(* IEC 61131-3 sources: website/app/projektit/rau-tyokalut/modbusrajapinta/examples/Common_functions, 30 files *)

(* ---- bitClearF.ST ---- *)
FUNCTION bitClearF : BOOL
VAR_INPUT
bitString : word;
bitNumber : uint;
END_VAR

VAR
bResult : bool;
wTemp : word;
END_VAR
(************************************************************)
(*	Function checks if bit is cleared in given bit string 	*)
(*															*)
(*	Inputs: bitString as 16bit word							*)
(*			bitNumber as unsigned integer from 0 to 15		*)
(*	Returns: Boolean value							  		*)
(*	Use: if bitClearF(bitString, bitNumber) then	 	  	*)
(*				do_something();						  		*)
(*		 end_if;											*)
(*													  		*)
(************************************************************)

if bitNumber > 15 then
	bResult := false;
else
	wTemp := 1;
	wTemp := SHL(wTemp, bitNumber);
	bResult := (bitString AND wTemp) = 0;
end_if;
bitClearF := bResult;

END_FUNCTION

(* ---- bitSetF.ST ---- *)
FUNCTION bitSetF : BOOL
VAR_INPUT
bitString : word;
bitNumber : uint;
END_VAR

VAR
bResult : bool;
wTemp : word;
END_VAR
(************************************************************)
(*	Function checks if bit is set in given bit string 		*)
(*															*)
(*	Inputs: bitString as 16bit word							*)
(*			bitNumber as unsigned integer from 0 to 15		*)
(*	Returns: Boolean value							  		*)
(*	Use: if bitSetF(bitString, bitNumber) then	 	  		*)
(*				do_something();						  		*)
(*		 end_if;											*)
(*													  		*)
(************************************************************)

if bitNumber > 15 then
	bResult := false;
else
	wTemp := 1;
	wTemp := SHL(wTemp, bitNumber);
	bResult := (bitString AND wTemp) > 0;
end_if;
bitSetF := bResult;

END_FUNCTION

(* ---- clearBitF.ST ---- *)
FUNCTION clearBitF : WORD
VAR_INPUT
bitString : word;
bitNumber : uint;
END_VAR

VAR
wResult : word;
wTemp : word;
END_VAR
(************************************************************)
(*	Function clears bit in given bit string 				*)
(*															*)
(*	Inputs: bitString as 16bit word							*)
(*			bitNumber as unsigned integer from 0 to 15		*)
(*	Returns: bitString with the bit cleared as 16bit word  	*)
(*	Use: bitString:=clearBitF(bitString, bitNumber);	 	*)
(*													  		*)
(************************************************************)

if bitNumber > 15 then
	wResult := bitString;
else
	wTemp := 1;
	wTemp := SHL(wTemp, bitNumber);
	wResult := bitString AND (16#FFFF XOR wTemp);
end_if;
clearBitF := wResult;

END_FUNCTION

(* ---- CoilF.ST ---- *)
FUNCTION CoilF : WORD
VAR_INPUT
	id_String : string(30);
	RegValue : word;
	BitMask : word;
END_VAR

VAR
	iTemp : int;
	iLockState : int;
	bFX2020 : bool;
	bReg : bool;
	ReturnValue : word;
END_VAR

bFX2020 := INT_TO_BOOL(GetDigitalPointF(Name:=id_String));
bReg:=WORD_TO_BOOL(RegValue AND BitMask);
iLockState:=GetLockStateF(Name:=id_String);

ReturnValue := RegValue;
IF id_String <> '' THEN
	if bFX2020 = bReg then
		(* Same value -> release manual override *)
		iTemp:=SetDigitalPointF(Value:=BOOL_TO_INT(bReg), LockState := 3, Name := id_String);
	elsif (iLockState = 2 or iLockState = 12) then
		(* The value have been changed in FX *)
		if (bFX2020 = true) then
			ReturnValue := (RegValue OR BitMask);
		else
			ReturnValue := (RegValue AND NOT(BitMask));
		end_if;
	else
		(* The value may have been changed in handterminal *)
	 	iTemp:=SetDigitalPointF(Value:=BOOL_TO_INT(bReg), LockState := 1, Name := id_String);
	end_if;
END_IF;

CoilF := ReturnValue;

END_FUNCTION

(* ---- CoilF_2.ST ---- *)
FUNCTION CoilF_2 : WORD
VAR_INPUT
	id_String : string(30);
	RegValue : word;
	BitMask : word;
	force : int;
END_VAR

VAR
	iTemp : int;
	iLockState : int;
	bFX2020 : bool;
	bReg : bool;
	ReturnValue : word;
END_VAR
(*Different version of the CoilF-function, added a new input parameter 'force' that indicates if the value is wanted to be
 forced from FX to the modbus device 0 = no forcing, 1 = value is forced *)

bFX2020 := INT_TO_BOOL(GetDigitalPointF(Name:=id_String));
bReg:=WORD_TO_BOOL(RegValue AND BitMask);
iLockState:=GetLockStateF(Name:=id_String);

ReturnValue := RegValue;
IF id_String <> '' THEN
	if bFX2020 = bReg then
		(* Same value -> release manual override *)
		iTemp:=SetDigitalPointF(Value:=BOOL_TO_INT(bReg), LockState := 3, Name := id_String);
	elsif (iLockState = 2 or iLockState = 12 or force = 1) then
		(* The value have been changed in FX, or user wants to force the point from FX *)
		if (bFX2020 = true) then
			ReturnValue := (RegValue OR BitMask);
		else
			ReturnValue := (RegValue AND NOT(BitMask));
		end_if;
	else
		(* The value may have been change in handterminal *)
	 	iTemp:=SetDigitalPointF(Value:=BOOL_TO_INT(bReg), LockState := 1, Name := id_String);
	end_if;
END_IF;

CoilF_2 := ReturnValue;

END_FUNCTION

(* ---- CoilF_3.ST ---- *)
FUNCTION CoilF_3 : WORD
VAR_INPUT
	id_String : string(30);
	RegValue : word;
	BitMask : word;
	Force : bool;
	ReleaseOverride : bool;
END_VAR

VAR
	iTemp : int;
	iLockState : int;
	bFX2020 : bool;
	bReg : bool;
	ReturnValue : word;
END_VAR

bFX2020 := INT_TO_BOOL(GetDigitalPointF(Name:=id_String));
bReg:=WORD_TO_BOOL(RegValue AND BitMask);
iLockState:=GetLockStateF(Name:=id_String);

ReturnValue := RegValue;
IF id_String <> '' THEN
	if bFX2020 = bReg and releaseOverride = true then
		(* Same value -> release manual override *)
		iTemp:=SetDigitalPointF(Value:=BOOL_TO_INT(bReg), LockState := 3, Name := id_String);
	elsif (iLockState = 2 or iLockState = 12 or force = true) then
		(* The value have been changed in FX *)
		if (bFX2020 = true) then
			ReturnValue := (RegValue OR BitMask);
		else
			ReturnValue := (RegValue AND NOT(BitMask));
		end_if;
	else
		(* The value may have been changed in handterminal *)
	 	iTemp:=SetDigitalPointF(Value:=BOOL_TO_INT(bReg), LockState := 1, Name := id_String);
	end_if;
END_IF;

CoilF_3 := ReturnValue;

END_FUNCTION

(* ---- DiscreteInputF.ST ---- *)
FUNCTION DiscreteInputF : INT
VAR_INPUT
	id_String : string(30);
	RegValue : word;
	BitMask : word;
END_VAR

VAR
	tulos : int;
END_VAR

IF id_String <> '' THEN
	(* Check BitMask defined bit status *)
	tulos := SetDigitalPointF(Value:=BOOL_TO_INT(WORD_TO_BOOL(RegValue AND BitMask)), LockState:=1, Name:=id_String);
	DiscreteInputF := 0;
ELSE
	DiscreteInputF := 9999;
END_IF;

END_FUNCTION

(* ---- DOUBLEHOLDINGREGF.ST ---- *)
FUNCTION DOUBLEHOLDINGREGF : UDINT
VAR_INPUT
	id_String : string(30);
	HighRegValue : word;
	LowRegValue : word;
	rMultiplier : real;
END_VAR

VAR
	rMultiply : real;
	rFX2025 : real;
	rReg : real;
	iLockState : int;
	iTemp : int;
	iReg : int;
	udiConversion : udint;
	diConversion : dint;
	rconversion : real;
	Result : int;
END_VAR
(* Zero division not allowed *)
rMultiply := rMultiplier;
if (rMultiply = 0.0) then
	rMultiply := 1.0;
end_if;

(* Read current FX2025 value *)
rFX2025 := GetAnalogPointF(Name:=id_String);

(* Convert double register value to real value *)
udiConversion := 65536*WORD_TO_UDINT(HighRegValue) + WORD_TO_UDINT(LowRegValue);
diConversion := UDINT_TO_DINT(udiConversion);
rConversion := DINT_TO_REAL(diConversion)/rMultiply;

(* Check LockState *)
iLockState:=GetLockStateF(Name:=id_String);

if id_String <> '' then
	if (rFX2025 = rConversion) then
		(* Same value -> release manual override *)
		Result := SetAnalogPointF(Value:=rConversion, LockState:=3, Name:=id_String);
	elsif (iLockState = 2 or iLockState = 12) then
		(* The value have been changed in FX *)
		diConversion := REAL_TO_DINT(rFX2025 * rMultiply);
		udiConversion := DINT_TO_UDINT(diConversion);
	else
		(* The value may have been changed in modbus equipment *)
		Result := SetAnalogPointF(Value:=rConversion, LockState:=1, Name:=id_String);
	end_if;
end_if;

DoubleHoldingRegF := udiConversion;

END_FUNCTION

(* ---- DOUBLEHOLDINGREGF_3DINT.ST ---- *)
FUNCTION DOUBLEHOLDINGREGF_3DINT : UDINT
VAR_INPUT
	id_String : string(30);
	HighRegValue : word;
	LowRegValue : word;
	rMultiplier : real;
	Force : bool;
	ReleaseOverride : bool;
END_VAR

VAR
	rMultiply : real;
	rFX2025 : real;
	rReg : real;
	iLockState : int;
	iTemp : int;
	iReg : int;
	udiConversion : udint;
	diConversion : dint;
	rconversion : real;
	Result : int;
END_VAR
(* Zero division not allowed *)
rMultiply := rMultiplier;
if (rMultiply = 0.0) then
	rMultiply := 1.0;
end_if;

(* Read current FX2025 value *)
rFX2025 := GetAnalogPointF(Name:=id_String);

(* Convert double register value to real value *)
udiConversion := 65536*WORD_TO_UDINT(HighRegValue) + WORD_TO_UDINT(LowRegValue);
diConversion := UDINT_TO_DINT(udiConversion);
rConversion := DINT_TO_REAL(diConversion)/rMultiply;

(* Check LockState *)
iLockState:=GetLockStateF(Name:=id_String);

if id_String <> '' then
	if (rFX2025 = rConversion and ReleaseOverride = true) then
		(* Same value -> release manual override *)
		Result := SetAnalogPointF(Value:=rConversion, LockState:=3, Name:=id_String);
	elsif (iLockState = 2 or iLockState = 12 or Force = true) then
		(* The value have been changed in FX *)
		diConversion := REAL_TO_DINT(rFX2025 * rMultiply);
		udiConversion := DINT_TO_UDINT(diConversion);
	else
		(* The value may have been changed in modbus equipment *)
		Result := SetAnalogPointF(Value:=rConversion, LockState:=1, Name:=id_String);
	end_if;
end_if;

DoubleHoldingRegF_3DINT := udiConversion;

END_FUNCTION

(* ---- DOUBLEHOLDINGREGF_3UDINT.ST ---- *)
FUNCTION DOUBLEHOLDINGREGF_3UDINT : UDINT
VAR_INPUT
	id_String : string(30);
	HighRegValue : word;
	LowRegValue : word;
	rMultiplier : real;
	Force : bool;
	ReleaseOverride : bool;
END_VAR

VAR
	rMultiply : real;
	rFX2025 : real;
	rReg : real;
	iLockState : int;
	iTemp : int;
	iReg : int;
	udiConversion : udint;
	rconversion : real;
	Result : int;
END_VAR
(* Zero division not allowed *)
rMultiply := rMultiplier;
if (rMultiply = 0.0) then
	rMultiply := 1.0;
end_if;

(* Read current FX2025 value *)
rFX2025 := GetAnalogPointF(Name:=id_String);

(* Convert double register value to real value *)
udiConversion := 65536*WORD_TO_UDINT(HighRegValue) + WORD_TO_UDINT(LowRegValue);
rConversion := UDINT_TO_REAL(udiConversion)/rMultiply;

(* Check LockState *)
iLockState:=GetLockStateF(Name:=id_String);

if id_String <> '' then
	if (rFX2025 = rConversion and ReleaseOverride = true) then
		(* Same value -> release manual override *)
		Result := SetAnalogPointF(Value:=rConversion, LockState:=3, Name:=id_String);
	elsif (iLockState = 2 or iLockState = 12 or Force = true) then
		(* The value have been changed in FX *)
		udiConversion := REAL_TO_UDINT(rFX2025 * rMultiply);
	else
		(* The value may have been changed in modbus equipment *)
		Result := SetAnalogPointF(Value:=rConversion, LockState:=1, Name:=id_String);
	end_if;
end_if;

DoubleHoldingRegF_3UDINT := udiConversion;

END_FUNCTION

(* ---- DoubleHoldingRegF_EM.ST ---- *)
FUNCTION DoubleHoldingRegF_EM : UDINT
VAR_INPUT
	id_String : string(30);
	HighRegValue : word;
	LowRegValue : word;
	rMultiplier : real;
END_VAR

VAR
	rMultiply : real;
	rFX2025 : real;
	rReg : real;
	iLockState : int;
	iTemp : int;
	iReg : int;
	udiConversion : udint;
	diConversion : dint;
	rconversion : real;
	Result : int;
END_VAR
(* Zero division not allowed *)
rMultiply := rMultiplier;
if (rMultiply = 0.0) then
	rMultiply := 1.0;
end_if;

(* Read current FX2025 value *)
rFX2025 := GetAnalogPointF(Name:=id_String);

(* Convert double register value to real value *)
udiConversion := 65536*WORD_TO_UDINT(HighRegValue) + WORD_TO_UDINT(LowRegValue);
diConversion := UDINT_TO_DINT(udiConversion);
rConversion := DINT_TO_REAL(diConversion)/rMultiply;

(* Check LockState *)
iLockState:=GetLockStateF(Name:=id_String);

if id_String <> '' then
	if (rFX2025 = rConversion) then
		(* Same value -> release manual override *)
		Result := SetAnalogPointF(Value:=rConversion, LockState:=3, Name:=id_String);
	elsif (iLockState = 2 or iLockState = 12) then
		(* The value have been changed in FX *)
		(* Energiamittarin rekisterit voidaan vain nollata *)
		if (rFX2025 <> 0.0) then
			Result := SetAnalogPointF(Value:=rConversion, LockState:=3, Name:=id_String);
		else
			udiConversion := 0;
		end_if;
	else
		(* The value may have been changed in modbus equipment *)
		Result := SetAnalogPointF(Value:=rConversion, LockState:=1, Name:=id_String);
	end_if;
end_if;

DoubleHoldingRegF_EM := udiConversion;

END_FUNCTION

(* ---- DoubleHoldingRegF_FLOAT.ST ---- *)
FUNCTION DoubleHoldingRegF_FLOAT : DWORD
VAR_INPUT
	id_String : string(30);
	LowRegValue : word;
	HighRegValue : word;
END_VAR

VAR
	rFX2020 : real;
	rReg : real;
	iLockState : int;
	iTemp : int;
	iReg : int;
	dwArvo : dword;
	realArvo : real;
END_VAR
(*point value in Fx*)
rFX2020 := GetAnalogPointF(Name:=id_String);

(* Value from modbus *)
dwArvo := WORD_TO_DWORD( HighRegValue );  (* Muunnnos 32 bittiseksi *)
dwArvo := SHL( dwArvo, 16 );   (* Siirret??n 16 bitti? vasemmalle *)
dwArvo := dwArvo OR WORD_TO_DWORD( LowRegValue );   (* Lis?t??n alemmat 16 bitti? *)
realArvo := WORD2_TO_REAL( dwArvo )  ;   (* Muunnetaan REAL tyyppiseksi *)
iLockState:=GetLockStateF(Name:=id_String);

IF id_String <> '' THEN
	if rFX2020 = realArvo then
		(* Same value -> release manual override *)
		iTemp:=SetAnalogPointF(Value:=rReg, LockState := 3, Name := id_String);
	elsif (iLockState = 2 or iLockState = 12) then
		(* The value have been changed in FX *)
		realArvo := rFX2020;
		dwArvo := REAL_TO_WORD2(realArvo); (*modify the return value so that it can be written to registers*)
	else
		(* The value may have been change in handterminal *)
		iTemp:=SetAnalogPointF(Value:=realArvo, LockState := 1, Name := id_String);
	end_if;
END_IF;

(* return the register values in a DWORD*)
DoubleHoldingRegF_FLOAT := dwArvo;

END_FUNCTION

(* ---- DoubleInputReg_Float.ST ---- *)
FUNCTION DoubleInputReg_Float : REAL
VAR_INPUT
	id_String : string(30);
	HighRegValue : word;
	LowRegValue : word;
END_VAR

VAR
	dwArvo : dword;
	realArvo : real;
	result : int;
END_VAR

dwArvo := WORD_TO_DWORD( HighRegValue );  (* Muunnnos 32 bittiseksi *)
dwArvo := SHL( dwArvo, 16 );   (* Siirret??n 16 bitti? vasemmalle *)
dwArvo := dwArvo OR WORD_TO_DWORD( LowRegValue );   (* Lis?t??n alemmat 16 bitti? *)
realArvo := WORD2_TO_REAL( dwArvo )  ;   (* Muunnetaan REAL tyyppiseksi *)

(* Talletetaan arvo mittauspisteeseen *)
result := SetAnalogPointF( Value := realArvo , LockState:=1, Name:= id_String );

DoubleInputReg_Float := realArvo;

END_FUNCTION

(* ---- DoubleInputReg_Float_jakaja.ST ---- *)
FUNCTION DoubleInputReg_Float_jakaja : REAL
VAR_INPUT
	id_String : string(30);
	HighRegValue : word;
	LowRegValue : word;
	jakaja : real;
END_VAR

VAR
	dwArvo : dword;
	realArvo : real;
	result : int;
END_VAR

dwArvo := WORD_TO_DWORD( HighRegValue );  (* Muunnnos 32 bittiseksi *)
dwArvo := SHL( dwArvo, 16 );   (* Siirret??n 16 bitti? vasemmalle *)
dwArvo := dwArvo OR WORD_TO_DWORD( LowRegValue );   (* Lis?t??n alemmat 16 bitti? *)
realArvo := WORD2_TO_REAL( dwArvo )  ;   (* Muunnetaan REAL tyyppiseksi *)

if(jakaja > 0.0) then
	realArvo := realArvo / jakaja;
end_if;

(* Talletetaan arvo mittauspisteeseen *)
result := SetAnalogPointF( Value := realArvo , LockState:=1, Name:= id_String );

DoubleInputReg_Float_jakaja := realArvo;

END_FUNCTION

(* ---- DoubleInputReg_WM14.ST ---- *)
FUNCTION DoubleInputReg_WM14 : REAL
VAR_INPUT
	id_String : string(30);
	HighRegValue : word;
	LowRegValue : word;
END_VAR

VAR
	dwArvo : dword;
	realArvo : real;
	result : int;
END_VAR

dwArvo := WORD_TO_DWORD( HighRegValue );  (* Muunnnos 32 bittiseksi *)
dwArvo := SHL( dwArvo, 16 );   (* Siirret??n 16 bitti? vasemmalle *)
dwArvo := dwArvo OR WORD_TO_DWORD( LowRegValue );   (* Lis?t??n alemmat 16 bitti? *)
realArvo := WORD2_TO_REAL( dwArvo )  ;   (* Muunnetaan REAL tyyppiseksi *)

(* Talletetaan arvo mittauspisteeseen *)
result := SetAnalogPointF( Value := realArvo , LockState:=1, Name:= id_String );

DoubleInputReg_WM14 := realArvo;

END_FUNCTION

(* ---- DoubleInputRegF.ST ---- *)
FUNCTION DoubleInputRegF : UDINT
VAR_INPUT
	id_String : string(30);
	HighRegValue : word;
	LowRegValue : word;
	rMultiplier : real;
END_VAR

VAR
	rMultiply : real;
	rFX2025 : real;
	rReg : real;
	iLockState : int;
	iTemp : int;
	iReg : int;
	udiConversion : udint;
	diConversion : dint;
	rconversion : real;
	Result : int;
END_VAR
(* Zero division not allowed *)
rMultiply := rMultiplier;
if (rMultiply = 0.0) then
	rMultiply := 1.0;
end_if;

(* Convert double register value to real value *)
udiConversion := 65536*WORD_TO_UDINT(HighRegValue) + WORD_TO_UDINT(LowRegValue);
diConversion := UDINT_TO_DINT(udiConversion);
rConversion := DINT_TO_REAL(diConversion)/rMultiply;

(* Save value to point database *)
Result := SetAnalogPointF(Value:=rConversion, LockState:=1, Name:=id_String);

DoubleInputRegF := udiConversion;

END_FUNCTION

(* ---- DoubleInputRegF_DINT.ST ---- *)
FUNCTION DoubleInputRegF_DINT : UDINT
VAR_INPUT
	id_String : string(30);
	HighRegValue : word;
	LowRegValue : word;
	rMultiplier : real;
END_VAR

VAR
	rMultiply : real;
	rFX2025 : real;
	rReg : real;
	iLockState : int;
	iTemp : int;
	iReg : int;
	udiConversion : udint;
	diConversion : dint;
	rconversion : real;
	Result : int;
END_VAR
(* Zero division not allowed *)
rMultiply := rMultiplier;
if (rMultiply = 0.0) then
	rMultiply := 1.0;
end_if;

(* Convert double register value to real value *)
udiConversion := 65536*WORD_TO_UDINT(HighRegValue) + WORD_TO_UDINT(LowRegValue);
diConversion := UDINT_TO_DINT(udiConversion);
rConversion := DINT_TO_REAL(diConversion)/rMultiply;

(* Save value to point database *)
Result := SetAnalogPointF(Value:=rConversion, LockState:=1, Name:=id_String);

DoubleInputRegF_DINT := udiConversion;

END_FUNCTION

(* ---- DoubleInputRegF_UDINT.ST ---- *)
FUNCTION DoubleInputRegF_UDINT : UDINT
VAR_INPUT
	id_String : string(30);
	HighRegValue : word;
	LowRegValue : word;
	rMultiplier : real;
END_VAR

VAR
	rMultiply : real;
	rFX2025 : real;
	rReg : real;
	iLockState : int;
	iTemp : int;
	iReg : int;
	udiConversion : udint;
	rconversion : real;
	Result : int;
END_VAR
(* Zero division not allowed *)
rMultiply := rMultiplier;
if (rMultiply = 0.0) then
	rMultiply := 1.0;
end_if;

(* Convert double register value to real value *)
udiConversion := 65536*WORD_TO_UDINT(HighRegValue) + WORD_TO_UDINT(LowRegValue);
rConversion := UDINT_TO_REAL(udiConversion)/rMultiply;

(* Save value to point database *)
Result := SetAnalogPointF(Value:=rConversion, LockState:=1, Name:=id_String);

DoubleInputRegF_UDINT := udiConversion;

END_FUNCTION

(* ---- fxe_Input64F.ST ---- *)
FUNCTION fxe_Input64F :REAL
(*
PLC: Fidelix
Company: Fidelix Sverige AB
Created by: Åke Kindmark_PC2
Program: fxe_Input64F

Date		| Version	|Created under	| Changed by		| Remark
----------------------------------------------------------------------------
2021-10-07		|   		|OpenPCSv 7.1.5	| Åke Kindmark_PC2		|
*)
VAR_INPUT
	PointId						:STRING(30) := '';
	LowReg0Value				:WORD;
	LowReg1Value				:WORD;
	HighReg2Value				:WORD;
	HighReg3Value				:WORD;
	Options						:DWORD;
END_VAR

VAR
	LReg0Value					:WORD;
	LReg1Value					:WORD;
	HReg2Value					:WORD;
	HReg3Value					:WORD;
	L0_org						:WORD;
	L1_org						:WORD;
	H2_org						:WORD;
	H3_org						:WORD;
	byte1						:WORD;
	byte2						:WORD;
	byte3						:WORD;
	byte4						:WORD;
	byte5						:WORD;
	byte6						:WORD;
	byte7						:WORD;
	byte8						:WORD;
	L0_inv						:WORD;
	L1_inv						:WORD;
	H2_inv						:WORD;
	H3_inv						:WORD;
	rReg_0						:REAL;
	rReg_1						:REAL;
	rReg_2						:REAL;
	rReg_3						:REAL;
	rValue						:REAL;
	iResult						:INT;
	rMultiplier					:REAL;
	iAccess						:INT;
	iSize						:INT;
	bBitMask					:BOOL;
	bInvert						:BOOL;
	bEndian						:BOOL;
	bByte						:BOOL;
	bWord						:BOOL;
	bUnsigned					:BOOL;
END_VAR
(* Extract multiplier from options *)
CASE DWORD_TO_INT(7 AND SHR(Options, 13)) OF
	1: rMultiplier := 10.0;
	2: rMultiplier := 100.0;
	3: rMultiplier := 1000.0;
ELSE
	rMultiplier := 1.0;
END_CASE;

(* Extract access from options *)
iAccess := DWORD_TO_INT(3 AND Options);
(* Extract size from options *)
iSize := DWORD_TO_INT(SHR(Options, 11));
(* Extract bitmask flag from options *)
bBitMask := DWORD_TO_INT(16 AND Options) = 16;
(* Extract invert flag from options *)
bInvert := DWORD_TO_INT(32 AND Options) = 32;
(* Extract litle endian flag from options *)
bEndian := DWORD_TO_INT(64 AND Options) = 64;
(* Extract byte swap flag from options *)
bByte := DWORD_TO_INT(128 AND Options) = 128;
(* Extract word swap flag from options *)
bWord := DWORD_TO_INT(256 AND Options) = 256;
(* Extract unsigned flag from options *)
bUnsigned := DWORD_TO_INT(512 AND Options) = 512;

(* Read 64(4x16)-bits registervalue *)
LReg0Value := LowReg0Value;
LReg1Value := LowReg1Value;
HReg2Value := HighReg2Value;
HReg3Value := HighReg3Value;

(* Byteswap. Shift High(MSP) and Low(LSP) Bytes of each 16-bit register value? *)
IF bByte THEN
	(* Read the original value of the registers, the bytes of which are inverted *)
	L0_org := LReg0Value;
	L1_org := LReg1Value;
	H2_org := HReg2Value;
	H3_org := HReg3Value;
	(* Masking, followed by only the last 8 bits of the word *)
	byte1 := (L0_org AND 16#00FF);
	byte3 := (L1_org AND 16#00FF);
	byte5 := (H2_org AND 16#00FF);
	byte7 := (H3_org AND 16#00FF);
	(* Move the second byte to the first position, i.e. 8 bits to the left *)
	byte1 := SHL(byte1, 8);
	byte3 := SHL(byte3, 8);
	byte5 := SHL(byte5, 8);
	byte7 := SHL(byte7, 8);
	(* A new masking that leaves only the first byte and 8 zeros behind *)
	byte2 := (L1_org AND 16#FF00);
	byte4 := (H3_org AND 16#FF00);
	byte6 := (H3_org AND 16#FF00);
	byte8 := (H3_org AND 16#FF00);
	(* Move one byte to the right so that the 1st byte goes to the 2nd position *)
	byte2 := SHR(byte2, 8);
	byte4 := SHR(byte4, 8);
	byte6 := SHR(byte6, 8);
	byte8 := SHR(byte8, 8);
	(* Finally, the bytes are combined and the new value is written to the register *)
	L0_inv := (byte1 OR byte2);
	L1_inv := (byte3 OR byte4);
	h2_inv := (byte5 OR byte6);
	h3_inv := (byte7 OR byte8);
	LReg0Value := L0_inv;
	LReg1Value := L1_inv;
	HReg2Value := H2_inv;
	HReg3Value := H3_inv;
END_IF;

(* Wordswap. Shift Higher and Lower registers in 64-bits readout? *)
IF bWord THEN
	(* Shift reg value order, High -> Low *)
	rReg_0:=UINT_TO_REAL(WORD_TO_UINT(HReg3Value))* 65536.0 * 65536.0 * 65536.0;
	rReg_1:=UINT_TO_REAL(WORD_TO_UINT(HReg2Value))* 65536.0 * 65536.0;
	rReg_2:=UINT_TO_REAL(WORD_TO_UINT(LReg1Value))* 65536.0;
	rReg_3:=UINT_TO_REAL(WORD_TO_UINT(LReg0Value));
ELSE
	(* Normal 64-bits readout *)
	rReg_0:=UINT_TO_REAL(WORD_TO_UINT(LReg0Value))* 65536.0 * 65536.0 * 65536.0;
	rReg_1:=UINT_TO_REAL(WORD_TO_UINT(LReg1Value))* 65536.0 * 65536.0;
	rReg_2:=UINT_TO_REAL(WORD_TO_UINT(HReg2Value))* 65536.0;
	rReg_3:=UINT_TO_REAL(WORD_TO_UINT(HReg3Value));
END_IF;

IF PointId <> '' THEN
	(* Raw value*scaling *)
	rValue := (rReg_3 + rReg_2 + rReg_1 + rReg_0) * rMultiplier;

	(* Scaled value write to database *)
	iResult:= SetAnalogPointF(rValue, 1, PointId);

	fxe_Input64F := rValue;
ELSE
	fxe_Input64F := 9999.0;
END_IF;
END_FUNCTION

(* ---- HOLDINGREGF.ST ---- *)
FUNCTION HOLDINGREGF : WORD
VAR_INPUT
	id_String : string(30);
	RegValue : word;
	rMultiplier : real;
END_VAR

VAR
	rMultiply : real;
	rFX2020 : real;
	rReg : real;
	iLockState : int;
	iTemp : int;
	iReg : int;
END_VAR
(* Zero division not allowed *)
rMultiply := rMultiplier;
if (rMultiply = 0.0) then
	rMultiply := 1.0;
end_if;

rFX2020 := GetAnalogPointF(Name:=id_String);
(* WORD_TO_INT conversion needed because of possible negative values *)
iReg:=WORD_TO_INT(RegValue);
rReg:=INT_TO_REAL(iReg) / rMultiply;
iLockState:=GetLockStateF(Name:=id_String);

IF id_String <> '' THEN
	if rFX2020 = rReg then
		(* Same value -> release manual override *)
		iTemp:=SetAnalogPointF(Value:=rReg, LockState := 3, Name := id_String);
	elsif (iLockState = 2 or iLockState = 12) then
		(* The value have been changed in FX *)
		rReg := rFX2020;
	else
		(* The value may have been change in handterminal *)
		iTemp:=SetAnalogPointF(Value:=rReg, LockState := 1, Name := id_String);
	end_if;
END_IF;

(* REAL_TO_INT conversion needed because of possible negative values *)
iReg := REAL_TO_INT(rReg * rMultiply);
HoldingRegF := INT_TO_WORD(iReg);

END_FUNCTION

(* ---- HOLDINGREGF_3.ST ---- *)
FUNCTION HOLDINGREGF_3 : WORD
VAR_INPUT
	id_String : string(30);
	RegValue : word;
	rMultiplier : real;
	Force : bool;
	ReleaseOverride : bool;
END_VAR

VAR
	rMultiply : real;
	rFX2020 : real;
	rReg : real;
	iLockState : int;
	iTemp : int;
	iReg : int;
END_VAR
(* Zero division not allowed *)
rMultiply := rMultiplier;
if (rMultiply = 0.0) then
	rMultiply := 1.0;
end_if;

rFX2020 := GetAnalogPointF(Name:=id_String);
(* WORD_TO_INT conversion needed because of possible negative values *)
iReg:=WORD_TO_INT(RegValue);
rReg:=INT_TO_REAL(iReg) / rMultiply;
iLockState:=GetLockStateF(Name:=id_String);

IF id_String <> '' THEN
	if rFX2020 = rReg and releaseOverride = true then
		(* Same value -> release manual override *)
		iTemp:=SetAnalogPointF(Value:=rReg, LockState := 3, Name := id_String);
	elsif (iLockState = 2 or iLockState = 12 or force = true) then
		(* The value have been changed in FX *)
		rReg := rFX2020;
	else
		(* The value may have been change in handterminal *)
		iTemp:=SetAnalogPointF(Value:=rReg, LockState := 1, Name := id_String);
	end_if;
END_IF;

(* REAL_TO_INT conversion needed because of possible negative values *)
iReg := REAL_TO_INT(rReg * rMultiply);
HoldingRegF_3 := INT_TO_WORD(iReg);

END_FUNCTION

(* ---- HOLDINGREGF_3DINT.ST ---- *)
FUNCTION HOLDINGREGF_3DINT : WORD
VAR_INPUT
	id_String : string(30);
	RegValue : word;
	rMultiplier : real;
	Force : bool;
	ReleaseOverride : bool;
END_VAR

VAR
	rMultiply : real;
	rFX2020 : real;
	rReg : real;
	iLockState : int;
	iTemp : int;
	iReg : dint;
END_VAR
(* Zero division not allowed *)
rMultiply := rMultiplier;
if (rMultiply = 0.0) then
	rMultiply := 1.0;
end_if;

rFX2020 := GetAnalogPointF(Name:=id_String);
(* WORD_TO_INT conversion needed because of possible negative values *)
iReg:=WORD_TO_DINT(RegValue);
rReg:=DINT_TO_REAL(iReg) / rMultiply;
iLockState:=GetLockStateF(Name:=id_String);

IF id_String <> '' THEN
	if rFX2020 = rReg and releaseOverride = true then
		(* Same value -> release manual override *)
		iTemp:=SetAnalogPointF(Value:=rReg, LockState := 3, Name := id_String);
	elsif (iLockState = 2 or iLockState = 12 or force = true) then
		(* The value have been changed in FX *)
		rReg := rFX2020;
	else
		(* The value may have been change in handterminal *)
		iTemp:=SetAnalogPointF(Value:=rReg, LockState := 1, Name := id_String);
	end_if;
END_IF;

(* REAL_TO_INT conversion needed because of possible negative values *)
iReg := REAL_TO_DINT(rReg * rMultiply);
HoldingRegF_3dInt := DINT_TO_WORD(iReg);

END_FUNCTION

(* ---- HOLDINGREGF_3INT.ST ---- *)
FUNCTION HOLDINGREGF_3INT : WORD
VAR_INPUT
	id_String : string(30);
	RegValue : word;
	rMultiplier : real;
	Force : bool;
	ReleaseOverride : bool;
END_VAR

VAR
	rMultiply : real;
	rFX2020 : real;
	rReg : real;
	iLockState : int;
	iTemp : int;
	iReg : int;
END_VAR
(* Zero division not allowed *)
rMultiply := rMultiplier;
if (rMultiply = 0.0) then
	rMultiply := 1.0;
end_if;

rFX2020 := GetAnalogPointF(Name:=id_String);
(* WORD_TO_INT conversion needed because of possible negative values *)
iReg:=WORD_TO_INT(RegValue);
rReg:=INT_TO_REAL(iReg) / rMultiply;
iLockState:=GetLockStateF(Name:=id_String);

IF id_String <> '' THEN
	if rFX2020 = rReg and releaseOverride = true then
		(* Same value -> release manual override *)
		iTemp:=SetAnalogPointF(Value:=rReg, LockState := 3, Name := id_String);
	elsif (iLockState = 2 or iLockState = 12 or force = true) then
		(* The value have been changed in FX *)
		rReg := rFX2020;
	else
		(* The value may have been change in handterminal *)
		iTemp:=SetAnalogPointF(Value:=rReg, LockState := 1, Name := id_String);
	end_if;
END_IF;

(* REAL_TO_INT conversion needed because of possible negative values *)
iReg := REAL_TO_INT(rReg * rMultiply);
HoldingRegF_3Int := INT_TO_WORD(iReg);

END_FUNCTION

(* ---- HOLDINGREGF_3UINT.ST ---- *)
FUNCTION HOLDINGREGF_3DINT : WORD
VAR_INPUT
	id_String : string(30);
	RegValue : word;
	rMultiplier : real;
	Force : bool;
	ReleaseOverride : bool;
END_VAR

VAR
	rMultiply : real;
	rFX2020 : real;
	rReg : real;
	iLockState : int;
	iTemp : int;
	iReg : dint;
END_VAR
(* Zero division not allowed *)
rMultiply := rMultiplier;
if (rMultiply = 0.0) then
	rMultiply := 1.0;
end_if;

rFX2020 := GetAnalogPointF(Name:=id_String);
(* WORD_TO_INT conversion needed because of possible negative values *)
iReg:=WORD_TO_DINT(RegValue);
rReg:=DINT_TO_REAL(iReg) / rMultiply;
iLockState:=GetLockStateF(Name:=id_String);

IF id_String <> '' THEN
	if rFX2020 = rReg and releaseOverride = true then
		(* Same value -> release manual override *)
		iTemp:=SetAnalogPointF(Value:=rReg, LockState := 3, Name := id_String);
	elsif (iLockState = 2 or iLockState = 12 or force = true) then
		(* The value have been changed in FX *)
		rReg := rFX2020;
	else
		(* The value may have been change in handterminal *)
		iTemp:=SetAnalogPointF(Value:=rReg, LockState := 1, Name := id_String);
	end_if;
END_IF;

(* REAL_TO_INT conversion needed because of possible negative values *)
iReg := REAL_TO_DINT(rReg * rMultiply);
HoldingRegF_3uInt := DINT_TO_WORD(iReg);

END_FUNCTION

(* ---- InputRegF.ST ---- *)
FUNCTION InputRegF : INT
VAR_INPUT
	id_String : string(30);
	RegValue : word;
	rMultiplier : real;
END_VAR

VAR
	rMultiply : real;
	rReg : real;
	iReg : int;
	iTemp : int;
END_VAR
(* Zero division not allowed *)
rMultiply := rMultiplier;
if (rMultiply = 0.0) then
	rMultiply := 1.0;
end_if;

IF id_String <> '' THEN
	(* WORD_TO_INT conversion needed because of possible negative values *)
	iReg:=WORD_TO_INT(RegValue);
	rReg:=INT_TO_REAL(iReg) / rMultiply;
	iTemp := SetAnalogPointF(Value := rReg, LockState := 1, Name := id_String);
	InputRegF := 0;
ELSE
	InputRegF := 9999;
END_IF;

END_FUNCTION

(* ---- InputRegF_INT.ST ---- *)
FUNCTION InputRegF_INT : INT
VAR_INPUT
	id_String : string(30);
	RegValue : word;
	rMultiplier : real;
END_VAR

VAR
	rMultiply : real;
	rReg : real;
	iReg : int;
	iTemp : int;
END_VAR
(* Zero division not allowed *)
rMultiply := rMultiplier;
if (rMultiply = 0.0) then
	rMultiply := 1.0;
end_if;

IF id_String <> '' THEN
	(* WORD_TO_INT conversion needed because of possible negative values *)
	iReg:=WORD_TO_INT(RegValue);
	rReg:=INT_TO_REAL(iReg) / rMultiply;
	iTemp := SetAnalogPointF(Value := rReg, LockState := 1, Name := id_String);
	InputRegF_INT := 0;
ELSE
	InputRegF_INT := 9999;
END_IF;

END_FUNCTION

(* ---- InputRegF_UINT.ST ---- *)
FUNCTION InputRegF_UINT : INT
VAR_INPUT
	id_String : string(30);
	RegValue : word;
	rMultiplier : real;
END_VAR

VAR
	rMultiply : real;
	rReg : real;
	iReg : int;
	iTemp : int;
END_VAR

(* Zero division not allowed *)
rMultiply := rMultiplier;
if (rMultiply = 0.0) then
	rMultiply := 1.0;
end_if;

IF id_String <> '' THEN
	rReg:=WORD_TO_REAL(RegValue) / rMultiply;
	iTemp := SetAnalogPointF(Value := rReg, LockState := 1, Name := id_String);
	InputRegF_UINT := 0;
ELSE
	InputRegF_UINT := 9999;
END_IF;

END_FUNCTION

(* ---- ReadAndSetBitF.ST ---- *)
FUNCTION ReadAndSetBitF : WORD
VAR_INPUT
	id_string 			: String(30);
	RegValue 			: Word;
	BitNumber 			: uint;
	Force 				: bool;
	ReleaseOverride 	: bool;
END_VAR

VAR
	iFX2020 : int;
	iLockState : int;
	wTemp : Word;
	iReg : int;
	wReturn : word;

	iTemp : Int ;
	bitmask : word;
END_VAR

(* READS BIT FROM BIT STRING *)
wReturn := RegValue ;

if bitNumber <= 15 then

	iFX2020 := GetDigitalPointf( Name := ID_STRING );
	(* READ BIT VALUE *)
	bitmask :=  REAL_TO_WORD( 2.0 ** BitNumber) ;

	iReg := BOOL_TO_INT( WORD_TO_BOOL( RegValue AND BitMask ));

	(* READS LOCKSTATE *)
	iLockState:=GetLockStateF(Name:=id_String);

	IF id_String <> '' THEN
		if iFX2020 = iReg and releaseOverride = true then
			(* Same value -> release manual override *)
			iTemp:=SetDigitalPointF(Value:= iReg, LockState := 3, Name := id_String);
		elsif (iLockState = 2 or iLockState = 12 or force = true) then
			(* The value have been changed in FX *)
			(* rReg := rFX2020; *)
			(* The value have been changed in FX *)
			if (iFX2020 = 1) then

				wReturn := (RegValue OR bitmask);
			else
				wReturn := (RegValue AND NOT(BitMask));
			end_if;

		else
			(* The value may have been change in handterminal *)
			iTemp:=SetDigitalPointF(Value:=iReg, LockState := 1, Name := id_String);
		end_if;
	END_IF;

end_if;

ReadAndSetBitF := wReturn;

END_FUNCTION

(* ---- setBitF.ST ---- *)
FUNCTION setBitF : WORD
VAR_INPUT
bitString : word;
bitNumber : uint;
END_VAR

VAR
wResult : word;
wTemp : word;
END_VAR
(************************************************************)
(*	Function sets bit in given bit string 					*)
(*															*)
(*	Inputs: bitString as 16bit word							*)
(*			bitNumber as unsigned integer from 0 to 15		*)
(*	Returns: bitString with the bit set as 16bit word  		*)
(*	Use: bitString:=setBitF(bitString, bitNumber);	 		*)
(*													  		*)
(************************************************************)

if bitNumber > 15 then
	wResult := bitString;
else
	wTemp := 1;
	wTemp := SHL(wTemp, bitNumber);
	wResult := bitString OR wTemp;
end_if;
setBitF := wResult;

END_FUNCTION

(* ---- BYTE_SWAP.ST ---- *)
FUNCTION_BLOCK BYTE_SWAP
VAR_EXTERNAL

END_VAR

VAR_INPUT
word_orig : word;
END_VAR

VAR_OUTPUT
word_swapped : word;
END_VAR

VAR
	original : word := 0;
	inverted : word := 0;
	byte1, byte2 : word;
END_VAR
(*Blokki vaihtaa 2-tavuisen sanan tavujen paikkaa*)

(*Input: 16-bittinen sana*)
(*Output: input tavut k??nnettyn?, alkuper?iset bitit 1-8 paikoilla 9-16 ja p?invastoin*)

	(*Luetaan alkuper?inen rekisterin arvo, jonka tavut k??nnet??n*)
	original := word_orig;

	(*Maskaus, jonka j?lkeen sanassa on vain 8 viimeist? bitti?*)
	byte1 := (original AND 16#00FF);

	(*Siirret??n toinen tavu ensimm?isen paikalle, eli 8 bitti? vasemmalle*)
	byte1 := SHL(byte1, 8);

	(*Uusi maskaus, jossa j?tet??n vain ensimm?inen tavu ja 8 nollaa per??n*)
	byte2 := (original AND 16#FF00);

	(*Siirret??n tavun verran oikealle, jolloin 1. tavu menee 2. paikalle*)
	byte2 := SHR(byte2, 8);

	(*Lopuksi yhdistet??n tavut ja kirjoitetaan uusi arvo rekisteriin*)
	inverted := (byte1 OR byte2);

	word_swapped := inverted;

END_FUNCTION_BLOCK
